FUNCTION_BLOCK ABSTRACT FB_AbstructAsset IMPLEMENTS I_Asset
VAR CONSTANT
	MAX_TEMPLATE_JOBS : UDINT := 10;
END_VAR
VAR_INPUT
END_VAR
VAR_OUTPUT
END_VAR
VAR
	_driver		: I_Container;
	_template_jobs : ARRAY [1..MAX_TEMPLATE_JOBS] OF I_JobCatalogue;
	_num_of_jobs : UDINT;
	_batch_job   : FB_Executor;
	_selected_process_job 		: I_JOB;
	_error_id : HRESULT;
	_asset_kind : E_AssetKind := E_AssetKind.station;
	_asset_name : STRING;
END_VAR

(* This is the generator that iteratively generates references to FB_executor instances*)
METHOD _index_generator_ : UINT;
VAR_INPUT
END_VAR
VAR_INST
	_init	: BOOL := FALSE;
	_current_order_number : UINT; // Represent order number of iteration
	_index: UINT;
END_VAR
IF NOT _init THEN
	_current_order_number := 0;
	_index := 1;
	_index_generator_ := 0;
	_init := TRUE;
END_IF

IF _num_of_jobs = 0 THEN
	RETURN;
END_IF


IF _current_order_number >= _num_of_jobs OR _index > MAX_TEMPLATE_JOBS THEN
	_init := FALSE;
END_IF

IF _init THEN
	WHILE _index < MAX_TEMPLATE_JOBS AND _template_jobs[_index] = 0 DO
		_index := _index + 1;
	END_WHILE
	IF _template_jobs[_index] <> 0 THEN
		_index_generator_ := _index;
	ELSE
		_index_generator_ := 0;
	END_IF
	_current_order_number := _current_order_number + 1;
	_index := _index + 1;
ELSE
	_index_generator_ := 0;
END_IF
END_METHOD

METHOD add_template_job : BOOL
VAR_INPUT
	template_job	: I_JobCatalogue;
END_VAR
VAR
	i : UDINT;
END_VAR
FOR i := 1 TO MAX_TEMPLATE_JOBS DO
	IF _template_jobs[i] = 0 THEN
		IF template_job.build_template_job() THEN
			_template_jobs[i] := template_job;
			_error_id := S_OK;
			add_template_job := TRUE;
			_num_of_jobs := _num_of_jobs + 1;
			RETURN;
		END_IF
	END_IF
END_FOR
_error_id := -1;
add_template_job := TRUE;
END_METHOD

PROPERTY asset_kind : E_AssetKind
GET
asset_kind := _asset_kind;
END_GET
SET
_asset_kind := asset_kind ;
END_SET
END_PROPERTY

PROPERTY asset_name : STRING
GET
asset_name := _asset_name;
END_GET
SET
_asset_name := asset_name;
_batch_job.future.future_name := _asset_name;
END_SET
END_PROPERTY

METHOD asset_start : BOOL
VAR_INPUT
END_VAR
IF _batch_job.ready THEN
	_batch_job.start();	
	asset_start := TRUE;
ELSE
	asset_start := FALSE;
END_IF
END_METHOD

PROPERTY driver : I_Job
SET
END_SET
END_PROPERTY

PROPERTY error_id : HRESULT
GET
error_id := _error_id;
END_GET
END_PROPERTY

//FB_Init is always available implicitly and it is used primarily for initialization.
//The return value is not evaluated. For a specific influence, you can also declare the
//methods explicitly and provide additional code there with the standard initialization
//code. You can evaluate the return value.
METHOD FB_Init: BOOL
VAR_INPUT
    bInitRetains: BOOL; // TRUE: the retain variables are initialized (reset warm / reset cold)
    bInCopyCode: BOOL;  // TRUE: the instance will be copied to the copy code afterward (online change)   
	driver : I_Container;
END_VAR
_batch_job.create_container(ContainerType.QUEUE, '');
_batch_job.continuous_mode := TRUE;
_batch_job.children.auto_start := FALSE;
IF driver = 0 THEN
	_error_id := -100;
	RETURN;
END_IF
_driver := driver;
_driver.append_job(_batch_job);
END_METHOD

PROPERTY iter_process_jobs : I_JobCatalogue
GET
VAR_INST
	_index : UDINT := 1;
END_VAR
_index := _index_generator_();
IF _index > 0 THEN
	IF _template_jobs[_index] <> 0 THEN
		IF _template_jobs[_index] <> 0 THEN
			iter_process_jobs := _template_jobs[_index];
		ELSE
			iter_process_jobs := 0;
		END_IF
	END_IF
ELSE
	iter_process_jobs := 0;
END_IF
END_GET
END_PROPERTY

METHOD process_job_start : BOOL
IF _selected_process_job = 0 THEN
	process_job_start := TRUE;
	_error_id := -1;
	RETURN;
END_IF
_batch_job.children.append_job(_selected_process_job);
_error_id := S_OK;
process_job_start := TRUE;
END_METHOD

{warning 'Add method implementation '}
METHOD remove_template_job_by_name : BOOL
VAR_INPUT
	template_name	: T_MaxString;
END_VAR
VAR
	i : UDINT;
END_VAR
FOR i := 1 TO MAX_TEMPLATE_JOBS DO
	IF _template_jobs[i].template_name = template_name THEN
		_template_jobs[i] := 0;
		_error_id := S_OK;
		remove_template_job_by_object := TRUE;
		RETURN;
	END_IF
END_FOR
_error_id := -2;
remove_template_job_by_object := TRUE;
END_METHOD

METHOD remove_template_job_by_object : BOOL
VAR_INPUT
	template_job	: I_Job;
END_VAR
VAR
	i : UDINT;
END_VAR
FOR i := 1 TO MAX_TEMPLATE_JOBS DO
	IF _template_jobs[i].template_job_object = _template_jobs THEN
		_template_jobs[i] := 0;
		_error_id := S_OK;
		remove_template_job_by_object := TRUE;
		_num_of_jobs := _num_of_jobs - 1;
		RETURN;
	END_IF
END_FOR
_error_id := -2;
remove_template_job_by_object := TRUE;
END_METHOD

METHOD select_process_job : BOOL
VAR_INPUT
	template_name : T_MaxString;
END_VAR
VAR
	job_template : I_JobCatalogue;
END_VAR
_error_id := -9;
REPEAT
	job_template := THIS^.iter_process_jobs;
	IF job_template <> 0 AND_THEN job_template.template_name = template_name THEN
		_selected_process_job := job_template.template_job_object;
		_error_id := S_OK;
	END_IF
UNTIL
	job_template = 0
END_REPEAT

select_process_job := TRUE;
END_METHOD

{warning 'Add property implementation'}
PROPERTY selected_process_job : I_Job
GET
selected_process_job := _selected_process_job;
END_GET
END_PROPERTY

{warning 'Add method implementation '}
METHOD set_parameters : BOOL
END_METHOD

END_FUNCTION_BLOCK

(* stored: Version 1.1.0.1, ProductVersion 3.1.4026.17
   POU FB_AbstructAsset: Id {d4d0355c-79fc-4600-bee5-c78f62e48799}, SpecialFunc None
   Method _index_generator_: Id {974a4970-f4cf-4e24-a956-ee0217ceeab4}
   Method add_template_job: Id {4358ad89-b831-401e-97f7-5b72f8b20c6f}
   Property asset_kind: Id {2ac5f7ca-9796-4b79-8958-254a0b97c0d0}
   Get Get: Id {0c768923-5fe9-4f39-9d49-438ae72e0815}
   Set Set: Id {649a0f38-de96-482a-bbc4-dd9f61c67234}
   Property asset_name: Id {3afe87e4-af7e-4675-b6b4-86d7284aa59a}
   Get Get: Id {9d1f333d-982d-4fcc-ab2a-85204f429608}
   Set Set: Id {0dc94d7a-169b-44ec-adc3-e1e3866e5821}
   Method asset_start: Id {66f78847-43f0-4d96-8ae7-3ddd2bcdbbec}
   Property driver: Id {cab1a5f0-3d1e-4843-a677-06939ef7a5ae}
   Set Set: Id {b5125617-136d-4390-a8bb-2e0d72edc21d}
   Property error_id: Id {7a356971-588c-4218-b502-06b7edd477a1}
   Get Get: Id {06f4107d-7cae-408c-9d3b-30afd98daf5a}
   Method FB_Init: Id {21cee4a2-3874-4f37-96ac-b683cedadefa}
   Property iter_process_jobs: Id {b94bd61e-9e02-46f0-bbcc-25c594961268}
   Get Get: Id {17f796f5-0748-4bce-9d9f-f1d25310a16c}
   Method process_job_start: Id {f7baef1b-480f-42d3-9246-dd99ce0e32ce}
   Method remove_template_job_by_name: Id {92eecbd9-ae24-4ab4-bbe7-285e5a8204ba}
   Method remove_template_job_by_object: Id {61c905ac-e7e2-4623-bb53-9dad92657542}
   Method select_process_job: Id {952130f9-79a5-406f-adc7-5c023024fd68}
   Property selected_process_job: Id {8b6d2da2-21cf-48f4-a563-68ecc4301090}
   Get Get: Id {c10ddf3f-e541-4ec8-ad36-ef73804d3a15}
   Method set_parameters: Id {e09870f8-3242-492f-9edb-7fb09b9795e8} *)
